PROGRAM MAIN
VAR
	dtTimestamp : DATE_AND_TIME := DT#2017-04-04-12:42:42;
  	(* JSON document *)
	fbJson 		: FB_JsonSaxWriter;
	sJsonDoc 	: STRING(255);
END_VAR

fbJson.StartObject();
fbJson.AddKey('Values');
fbJson.StartObject();
fbJson.AddKey('Timestamp');
fbJson.AddDateTime(dtTimestamp);
fbJson.AddKey('Sensor1');
fbJson.AddReal(42.42);
fbJson.AddKey('Sensor2');
fbJson.AddDint(42);
fbJson.AddKey('Sensor3');
fbJson.AddBool(TRUE);
fbJson.EndObject();
fbJson.EndObject();
sJsonDoc := fbJson.GetDocument();
fbJson.ResetDocument();

END_PROGRAM

(* stored: Version 1.1.0.1, ProductVersion 3.1.4021.12
   POU MAIN: Id {88652892-e7f6-4c6b-90e1-af4abe0f72ff}, SpecialFunc None *)
